// Mitsubishi GX Works2 project: Group_4   PLC: FX3G

// global labels: Global1
VAR_GLOBAL
  LightWork AT Y007 : BOOL;
  StartDay AT X007 : BOOL;
  EmergencyBut AT X011 : BOOL;
  StartCooking AT X001 : BOOL;
END_VAR
VAR_GLOBAL CONSTANT
  Lager : REAL := 5;
END_VAR
VAR_GLOBAL
  StartStockYeast AT D1101 : REAL;
  StockYeast AT D1103 : REAL;
  StartStockMalt AT D1105 : REAL;
  StockMalt AT D1107 : REAL;
  StartStockHops AT D1109 : REAL;
  StockHops AT D1111 : REAL;
END_VAR
VAR_GLOBAL CONSTANT
  MinYeast : REAL := 150;
  MinMalt : REAL := 12;
  MinHops : REAL := 60;
END_VAR
VAR_GLOBAL
  EnoughYeast AT M0 : BOOL;
  EnoughMalt AT M1 : BOOL;
  EnoughHops AT M2 : BOOL;
END_VAR
VAR_GLOBAL CONSTANT
  Pilzner : REAL := 6;
  MinYeastP : REAL := 150;
  MinYeastL : REAL := 150;
  MinMaltL : REAL := 12;
  MinMaltP : REAL := 6;
  MinHopsP : REAL := 53;
  MinHopsL : REAL := 60;
END_VAR
VAR_GLOBAL
  Y1Controler AT M3 : BOOL;
  CookingTime AT Y001 : BOOL;
  cook AT TC19 : BOOL;
END_VAR
VAR_GLOBAL CONSTANT
  CookDest : INT := 4000;
END_VAR
VAR_GLOBAL
  cookFinish AT TS19 : BOOL;
  LagerBulb AT M10 : BOOL;
  PilznerBulb AT M11 : BOOL;
  HelpM12 AT M12 : BOOL;
  HelpLight AT M12 : BOOL;
  HelpLight10 AT M12 : BOOL;
  HelpLight11 AT M12 : BOOL;
  AnalogAsFloat AT D1221 : REAL;
END_VAR
VAR_GLOBAL CONSTANT
  Divider : REAL := 400;
END_VAR
VAR_GLOBAL
  AnalogInput1 AT D8280 : INT;
  SaveAnalog1 AT D8201 : INT;
  cookTimerAnswer AT TS19 : BOOL;
  StartFermentation AT X005 : BOOL;
END_VAR
VAR_GLOBAL CONSTANT
  LagerFerm3Sec : INT := 3000;
  PilzFerm4Sec : INT := 4000;
END_VAR
VAR_GLOBAL
  FermTimer AT D1323 : INT;
  Light4 AT M4 : BOOL;
  FirstLightT21 AT TC21 : BOOL;
  Tss21 AT TS21 : BOOL;
  FirstLightAnswer AT TS21 : BOOL;
  FirstLightFerm AT Y003 : BOOL;
  SecondLightFerm AT Y004 : BOOL;
  SecondLightAnswer AT TS23 : BOOL;
  SecondLightT23 AT TC23 : BOOL;
  StartStorage AT X002 : BOOL;
  countBottle AT CC1 : BOOL;
END_VAR
VAR_GLOBAL CONSTANT
  SixBottle : INT := 5;
END_VAR
VAR_GLOBAL
  countSix AT CC2 : BOOL;
  StorageSix AT D1115 : REAL;
END_VAR
VAR_GLOBAL CONSTANT
  OneSix : REAL := 1;
END_VAR
VAR_GLOBAL
  OneBottle AT X000 : BOOL;
  FirstC1 AT CC1 : BOOL;
  LightStorage AT Y002 : BOOL;
  StorageLight AT Y002 : BOOL;
  CountFirstBottle AT CC2 : BOOL;
END_VAR
VAR_GLOBAL CONSTANT
  FirstBottle : REAL := 1;
END_VAR
VAR_GLOBAL
  FinishPacking AT M5 : BOOL;
END_VAR

// task Task_01 (event TRUE, interval 0, priority 31): POU_01

PROGRAM POU_01
(* structured ladder/FBD written out as ST: instructions are called as NAME(EN, inputs, outputs); _pN, _eN, _tN stand for wires *)
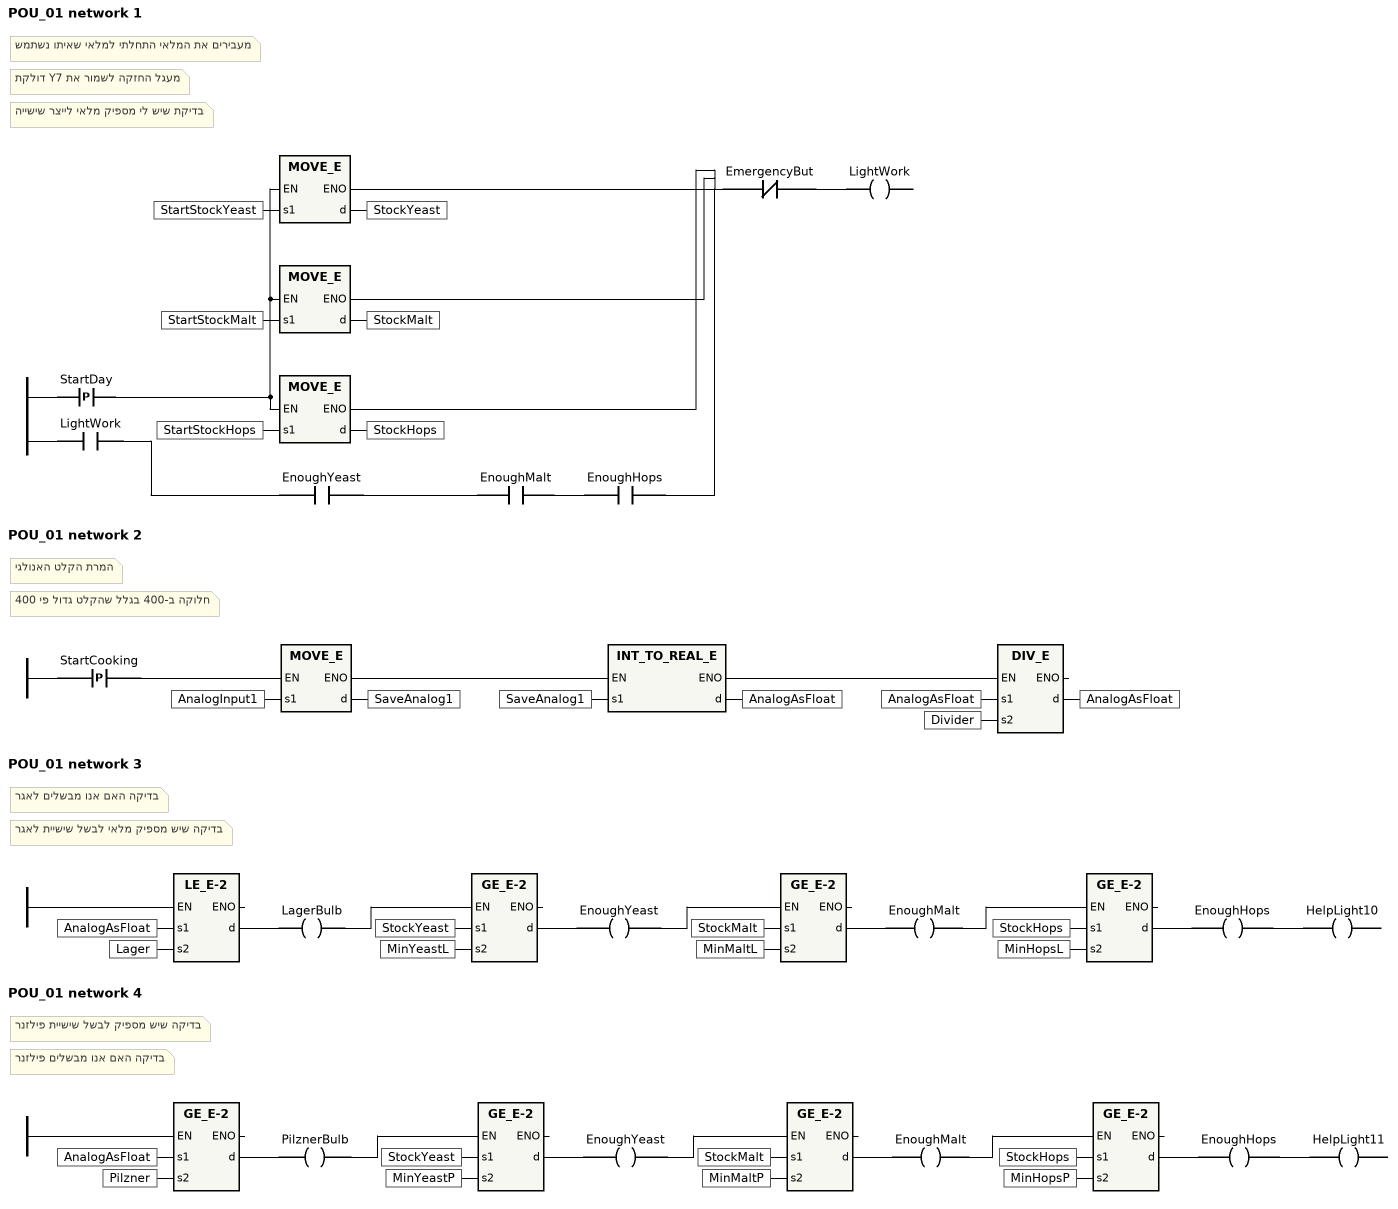
(* network 1 Day Init *)
(* מעבירים את המלאי התחלתי למלאי שאיתו נשתמש *)
(* מעגל החזקה לשמור את Y7 דולקת *)
(* בדיקת שיש לי מספיק מלאי לייצר שישייה *)
_p1 := LDP(TRUE, StartDay);
_e2 := MOVE_E(_p1, StartStockYeast, StockYeast);
_e3 := MOVE_E(_p1, StartStockMalt, StockMalt);
_e4 := MOVE_E(_p1, StartStockHops, StockHops);
LightWork := (_e2 OR _e3 OR _e4 OR (LightWork AND EnoughYeast AND EnoughMalt AND EnoughHops)) AND NOT EmergencyBut;
(* network 2 StartCook *)
(* המרת הקלט האנולגי *)
(* חלוקה ב-400 בגלל שהקלט גדול פי 400 *)
_e1 := MOVE_E(LDP(TRUE, StartCooking), AnalogInput1, SaveAnalog1);
_e2 := INT_TO_REAL_E(_e1, SaveAnalog1, AnalogAsFloat);
DIV_E(_e2, AnalogAsFloat, Divider, AnalogAsFloat);
(* network 3 CookLage *)
(* בדיקה האם אנו מבשלים לאגר *)
(* בדיקה שיש מספיק מלאי לבשל שישיית לאגר *)
LE_E(TRUE, AnalogAsFloat, Lager, _t1);
LagerBulb := _t1;
GE_E(_t1, StockYeast, MinYeastL, _t2);
EnoughYeast := _t2;
GE_E(_t2, StockMalt, MinMaltL, _t3);
EnoughMalt := _t3;
GE_E(_t3, StockHops, MinHopsL, _t4);
EnoughHops := _t4;
HelpLight10 := _t4;
(* network 4 CookPilz *)
(* בדיקה שיש מספיק לבשל שישיית פילזנר *)
(* בדיקה האם אנו מבשלים פילזנר *)
GE_E(TRUE, AnalogAsFloat, Pilzner, _t1);
PilznerBulb := _t1;
GE_E(_t1, StockYeast, MinYeastP, _t2);
EnoughYeast := _t2;
GE_E(_t2, StockMalt, MinMaltP, _t3);
EnoughMalt := _t3;
GE_E(_t3, StockHops, MinHopsP, _t4);
EnoughHops := _t4;
HelpLight11 := _t4;
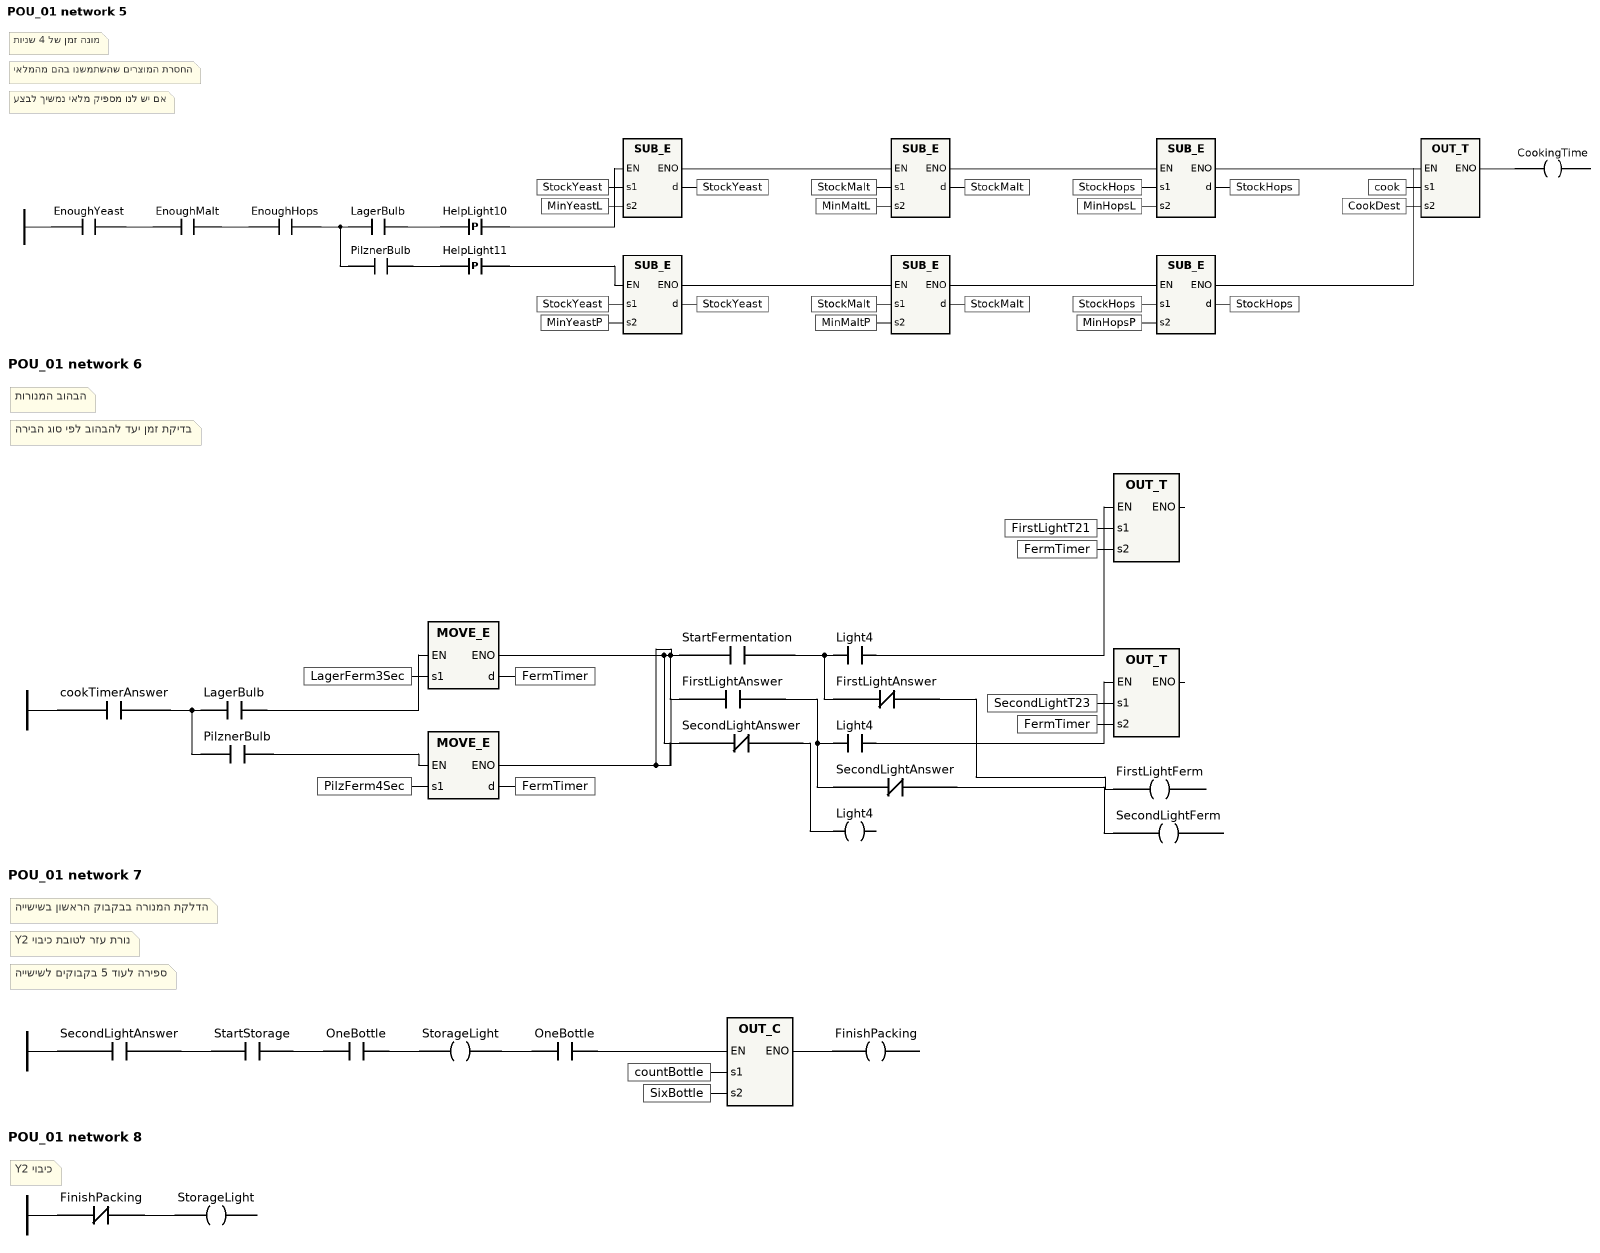
(* network 5 Cooking *)
(* מונה זמן של 4 שניות *)
(* החסרת המוצרים שהשתמשנו בהם מהמלאי *)
(* אם יש לנו מספיק מלאי נמשיך לבצע *)
_p1 := EnoughYeast AND EnoughMalt AND EnoughHops;
_e2 := SUB_E(_p1 AND LagerBulb AND LDP(TRUE, HelpLight10), StockYeast, MinYeastL, StockYeast);
_e3 := SUB_E(_e2, StockMalt, MinMaltL, StockMalt);
_e4 := SUB_E(_e3, StockHops, MinHopsL, StockHops);
_e5 := SUB_E(_p1 AND PilznerBulb AND LDP(TRUE, HelpLight11), StockYeast, MinYeastP, StockYeast);
_e6 := SUB_E(_e5, StockMalt, MinMaltP, StockMalt);
_e7 := SUB_E(_e6, StockHops, MinHopsP, StockHops);
_e8 := OUT_T(_e4 OR _e7, cook, CookDest);
CookingTime := _e8;
(* network 6 Fermentation *)
(* הבהוב המנורות *)
(* בדיקת זמן יעד להבהוב לפי סוג הבירה *)
_e1 := MOVE_E(cookTimerAnswer AND LagerBulb, LagerFerm3Sec, FermTimer);
_e2 := MOVE_E(cookTimerAnswer AND PilznerBulb, PilzFerm4Sec, FermTimer);
_p3 := _e1 OR _e2;
_p4 := _p3 AND StartFermentation;
OUT_T(_p4 AND Light4, FirstLightT21, FermTimer);
FirstLightFerm := _p4 AND NOT FirstLightAnswer;
_p5 := _p3 AND FirstLightAnswer;
OUT_T(_p5 AND Light4, SecondLightT23, FermTimer);
SecondLightFerm := _p5 AND NOT SecondLightAnswer;
Light4 := _p3 AND NOT SecondLightAnswer;
(* network 7 Storage *)
(* הדלקת המנורה בבקבוק הראשון בשישייה *)
(* נורת עזר לטובת כיבוי Y2 *)
(* ספירה לעוד 5 בקבוקים לשישייה *)
_p1 := SecondLightAnswer AND StartStorage AND OneBottle;
StorageLight := _p1;
_e2 := OUT_C(_p1 AND OneBottle, countBottle, SixBottle);
FinishPacking := _e2;
(* network 8 Turn_Off_Y2 *)
(* כיבוי Y2 *)
StorageLight := NOT FinishPacking;
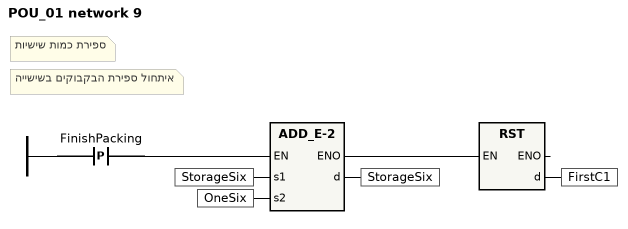
(* network 9 CountPackges *)
(* ספירת כמות שישיות *)
(* איתחול ספירת הבקבוקים בשישייה *)
_e1 := ADD_E(LDP(TRUE, FinishPacking), StorageSix, OneSix, StorageSix);
RST(_e1, FirstC1);
END_PROGRAM
